# EPICS alarm handler configuration: mps_database/bare/alarms/areas/mpln_l2b_mp04.alhConfig
GROUP NULL MPLN:L2B:MP04:1
$ALIAS MPS Link Node 64
$GUIDANCE
LTUH MPS
   Group Name: MPLN:L2B:MP04:1
   Summary PV:  MPLN:L2B:MP04:1:STATSUMY
$END
CHANNEL  MPLN:L2B:MP04:1    MPLN:L2B:MP04:1:MPS_EN_RBV		-----
CHANNEL  MPLN:L2B:MP04:1    MPLN:L2B:MP04:1:LC1_MODE_RBV		-----
